VAR_GLOBAL
	//Deck 1
	//Drive inputs
	ATV_State_D1							AT	%I*		: WORD; //Drive state
	ATV_TPDO_Input1_Status_Word_D1			AT	%I*		: WORD;	//Status Word From Drive
	iVelocityRaw_D1							AT	%I*		: INT;	//Velocity From Drive - Address 8604 - Units 1 RPM
	iTorqueRaw_D1							AT	%I*		: INT;	//Torque From Drive - Address 3205 - Units 0.1%
	uiCurrentRaw_D1							AT	%I*		: UINT;	//Current From Drive - Address 3204 - Units 0.1A
	uiVoltageRaw_D1							AT	%I*		: UINT;	//Voltage From Drive - Address 3208 - Units 1V
	uiFaultCode_D1							AT	%I*		: UINT;	//Fault Codes
	//End drive inputs	

	//Drive outputs
	ATV_RPDO_Output1_Control_Word_D1		AT	%Q*		: WORD;	//Control Word To Drive
	ATV_RPDO_Output2_Target_Velocity_D1		AT	%Q*		: WORD; //Velocity To Drive in RPM - Max Value 32767
	//End drive outputs

	//Inputs Status Word Bit Level
	xReady_To_Switch_on_D1 								: BOOL;//Bit 0
	xSwitched_ON_D1										: BOOL;//Bit 1
	xOperationEnabled_D1 								: BOOL;//Bit 2
	xFault_D1 											: BOOL;//Bit 3
	xVoltageEnabled_D1									: BOOL;//Bit 4
	xQuickStop_D1										: BOOL;//Bit 5
	xSwitchOnDisabled_D1 								: BOOL;//Bit 6
	xWarning_D1											: BOOL;//Bit 7
	xTargetReached_D1									: BOOL;//Bit 10
	xInternalLimitActive_D1								: BOOL;//Bit 11
	xDirectionofRotation_D1								: BOOL;//Bit 15	
	stFault_D1											: STRING;
	rTorqueValue_D1										: REAL;
	rCurrentValue_D1									: REAL;
	lrSpeed_D1											: LREAL;
	xEnable_D1											: BOOL; //Enable Drive Trigger
	xStart_D1											: BOOL;	//Start Trigger
	xStop_D1 											: BOOL;	//Stop Trigger
	iDirection_D1										: INT;	//Direction	Trigger
	xForward_D1											: BOOL; //Forward Trigger
	xReverse_D1											: BOOL;	//Reverse Trigger
	xReset_D1											: BOOL;	//Reset Trigger
	xInputStatus_HMI_D1									: ARRAY [0..9] OF BOOL;	//VFD Status Bits
	//End inputs Status Word Bit Level
	//End Deck 1
END_VAR

(* stored: Version 1.1.0.1, ProductVersion 3.1.4024.3
   GVL Deck1: Id {fb4fc70b-bfaf-49fd-86bb-866c5fb77624} *)
